INTERFACE I_MachineControl EXTENDS I_UniversalMachine

PROPERTY Robots : REFERENCE TO FB_CR800EtherCAT
GET
END_GET
END_PROPERTY

END_INTERFACE

(* stored: Version 1.1.0.1, ProductVersion 3.1.4024.9
   Itf I_MachineControl: Id {575cfd35-d864-4f94-b2bb-e1e7c6df6ebc}
   Property Robots: Id {508a7188-8eec-4c0a-b26d-0bdcd24ff2fb}
   Get Get: Id {eed6073b-58a6-4232-ab65-7b3da114e4ea} *)
